% RSLogix 500 project I2P-Hands-On 4 - Adam Boczkiewicz.RSS, saved by version 10.00.00.00 %
PROJECT "UNTITLED"    % processor: Bul.1763 MicroLogix 1100 Series B %

PROGRAM FILES
  LAD 2   15 rungs

DATA FILES
  O0 OUTPUT  4 elements
  I1 INPUT  6 elements
  S2 STATUS  66 elements
  B3 BINARY  1 elements
  T4 TIMER  1 elements
  C5 COUNTER  1 elements
  R6 CONTROL  1 elements
  N7 INTEGER  1 elements
  F8 FLOAT  1 elements

LADDER 2
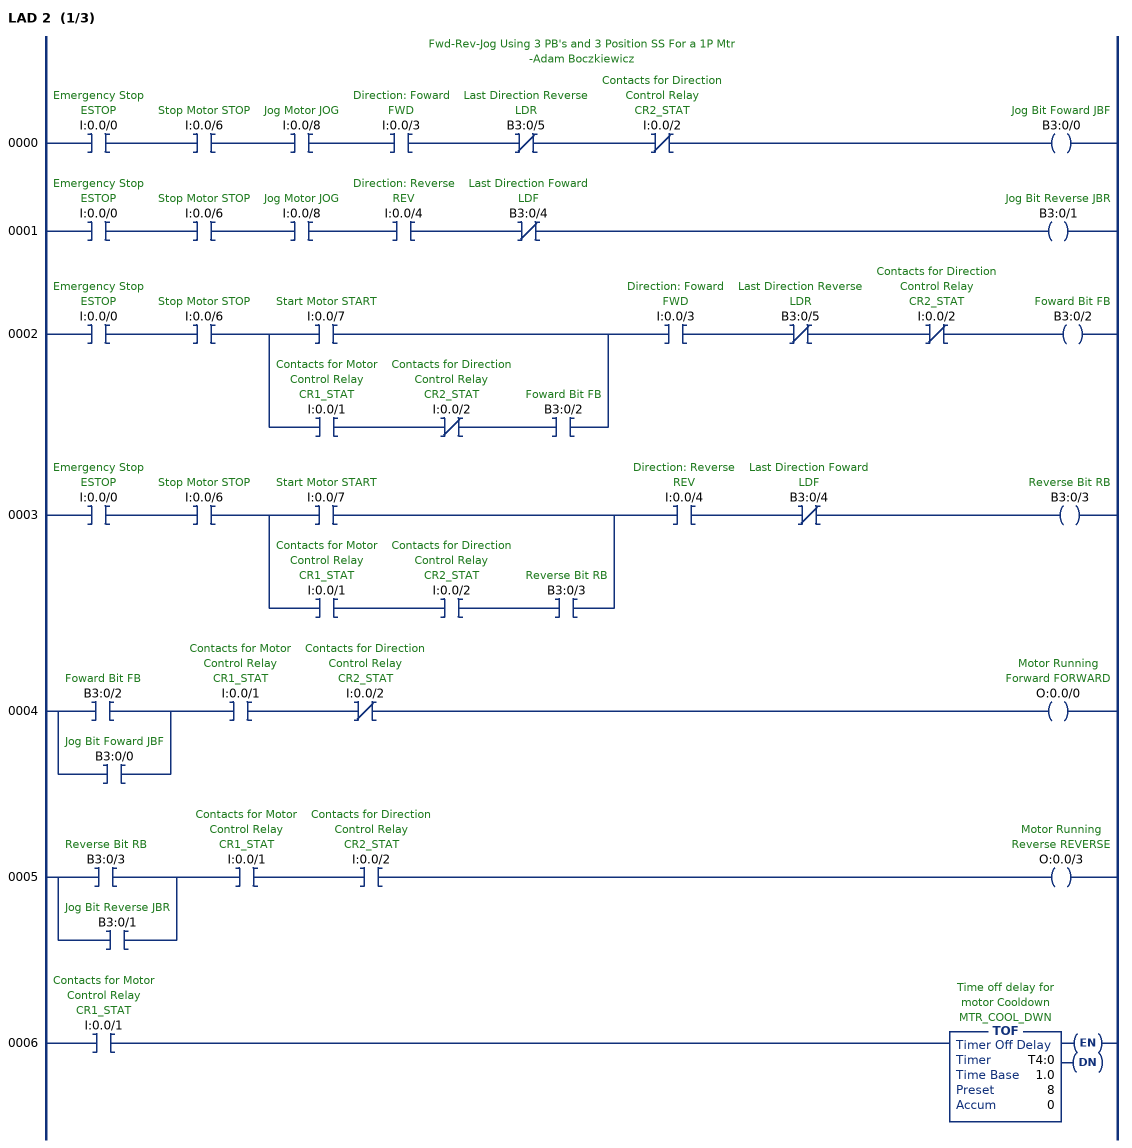
% Rung: 0 %
% Fwd-Rev-Jog Using 3 PB's and 3 Position SS For a 1P Mtr
% -Adam Boczkiewicz %
SOR XIC I:0.0/0 XIC I:0.0/6 XIC I:0.0/8 XIC I:0.0/3 XIO B3:0/5 XIO I:0.0/2 OTE B3:0/0 EOR
%   I:0.0/0  ESTOP  "Emergency Stop" %
%   I:0.0/6  STOP  "Stop Motor" %
%   I:0.0/8  JOG  "Jog Motor" %
%   I:0.0/3  FWD  "Direction: Foward" %
%   B3:0/5  LDR  "Last Direction Reverse" %
%   I:0.0/2  CR2_STAT  "Contacts for Direction Control Relay" %
%   B3:0/0  JBF  "Jog Bit Foward" %
% Rung: 1 %
SOR XIC I:0.0/0 XIC I:0.0/6 XIC I:0.0/8 XIC I:0.0/4 XIO B3:0/4 OTE B3:0/1 EOR
%   I:0.0/0  ESTOP  "Emergency Stop" %
%   I:0.0/6  STOP  "Stop Motor" %
%   I:0.0/8  JOG  "Jog Motor" %
%   I:0.0/4  REV  "Direction: Reverse" %
%   B3:0/4  LDF  "Last Direction Foward" %
%   B3:0/1  JBR  "Jog Bit Reverse" %
% Rung: 2 %
SOR XIC I:0.0/0 XIC I:0.0/6 BST XIC I:0.0/7 NXB XIC I:0.0/1 XIO I:0.0/2 XIC B3:0/2 BND XIC I:0.0/3 XIO B3:0/5 XIO I:0.0/2 OTE B3:0/2 EOR
%   I:0.0/0  ESTOP  "Emergency Stop" %
%   I:0.0/6  STOP  "Stop Motor" %
%   I:0.0/7  START  "Start Motor" %
%   I:0.0/1  CR1_STAT  "Contacts for Motor Control Relay" %
%   I:0.0/2  CR2_STAT  "Contacts for Direction Control Relay" %
%   B3:0/2  FB  "Foward Bit" %
%   I:0.0/3  FWD  "Direction: Foward" %
%   B3:0/5  LDR  "Last Direction Reverse" %
% Rung: 3 %
SOR XIC I:0.0/0 XIC I:0.0/6 BST XIC I:0.0/7 NXB XIC I:0.0/1 XIC I:0.0/2 XIC B3:0/3 BND XIC I:0.0/4 XIO B3:0/4 OTE B3:0/3 EOR
%   I:0.0/0  ESTOP  "Emergency Stop" %
%   I:0.0/6  STOP  "Stop Motor" %
%   I:0.0/7  START  "Start Motor" %
%   I:0.0/1  CR1_STAT  "Contacts for Motor Control Relay" %
%   I:0.0/2  CR2_STAT  "Contacts for Direction Control Relay" %
%   B3:0/3  RB  "Reverse Bit" %
%   I:0.0/4  REV  "Direction: Reverse" %
%   B3:0/4  LDF  "Last Direction Foward" %
% Rung: 4 %
SOR BST XIC B3:0/2 NXB XIC B3:0/0 BND XIC I:0.0/1 XIO I:0.0/2 OTE O:0.0/0 EOR
%   B3:0/2  FB  "Foward Bit" %
%   B3:0/0  JBF  "Jog Bit Foward" %
%   I:0.0/1  CR1_STAT  "Contacts for Motor Control Relay" %
%   I:0.0/2  CR2_STAT  "Contacts for Direction Control Relay" %
%   O:0.0/0  FORWARD  "Motor Running Forward" %
% Rung: 5 %
SOR BST XIC B3:0/3 NXB XIC B3:0/1 BND XIC I:0.0/1 XIC I:0.0/2 OTE O:0.0/3 EOR
%   B3:0/3  RB  "Reverse Bit" %
%   B3:0/1  JBR  "Jog Bit Reverse" %
%   I:0.0/1  CR1_STAT  "Contacts for Motor Control Relay" %
%   I:0.0/2  CR2_STAT  "Contacts for Direction Control Relay" %
%   O:0.0/3  REVERSE  "Motor Running Reverse" %
% Rung: 6 %
SOR XIC I:0.0/1 TOF T4:0 1.0 8 0 EOR
%   I:0.0/1  CR1_STAT  "Contacts for Motor Control Relay" %
%   T4:0  MTR_COOL_DWN  "Time off delay for motor Cooldown" %

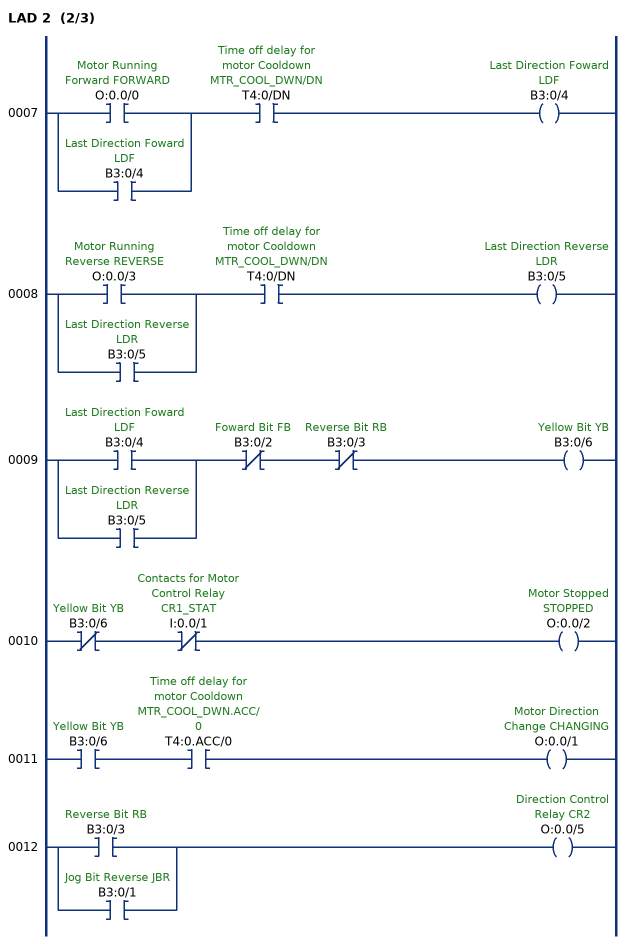
% Rung: 7 %
SOR BST XIC O:0.0/0 NXB XIC B3:0/4 BND XIC T4:0/DN OTE B3:0/4 EOR
%   O:0.0/0  FORWARD  "Motor Running Forward" %
%   B3:0/4  LDF  "Last Direction Foward" %
%   T4:0  MTR_COOL_DWN  "Time off delay for motor Cooldown" %
% Rung: 8 %
SOR BST XIC O:0.0/3 NXB XIC B3:0/5 BND XIC T4:0/DN OTE B3:0/5 EOR
%   O:0.0/3  REVERSE  "Motor Running Reverse" %
%   B3:0/5  LDR  "Last Direction Reverse" %
%   T4:0  MTR_COOL_DWN  "Time off delay for motor Cooldown" %
% Rung: 9 %
SOR BST XIC B3:0/4 NXB XIC B3:0/5 BND XIO B3:0/2 XIO B3:0/3 OTE B3:0/6 EOR
%   B3:0/4  LDF  "Last Direction Foward" %
%   B3:0/5  LDR  "Last Direction Reverse" %
%   B3:0/2  FB  "Foward Bit" %
%   B3:0/3  RB  "Reverse Bit" %
%   B3:0/6  YB  "Yellow Bit" %
% Rung: 10 %
SOR XIO B3:0/6 XIO I:0.0/1 OTE O:0.0/2 EOR
%   B3:0/6  YB  "Yellow Bit" %
%   I:0.0/1  CR1_STAT  "Contacts for Motor Control Relay" %
%   O:0.0/2  STOPPED  "Motor Stopped" %
% Rung: 11 %
SOR XIC B3:0/6 XIC T4:0.ACC/0 OTE O:0.0/1 EOR
%   B3:0/6  YB  "Yellow Bit" %
%   T4:0  MTR_COOL_DWN  "Time off delay for motor Cooldown" %
%   O:0.0/1  CHANGING  "Motor Direction Change" %
% Rung: 12 %
SOR BST XIC B3:0/3 NXB XIC B3:0/1 BND OTE O:0.0/5 EOR
%   B3:0/3  RB  "Reverse Bit" %
%   B3:0/1  JBR  "Jog Bit Reverse" %
%   O:0.0/5  CR2  "Direction Control Relay" %

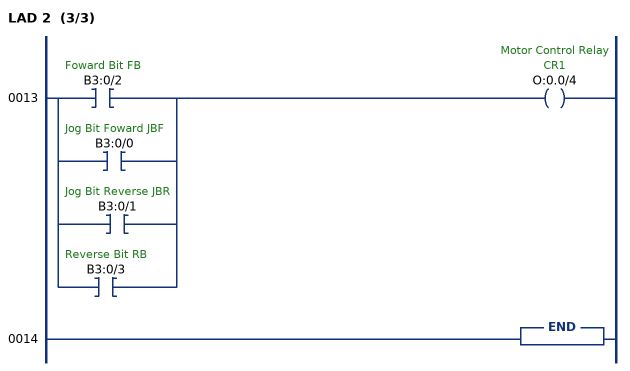
% Rung: 13 %
SOR BST XIC B3:0/2 NXB BST XIC B3:0/0 NXB BST XIC B3:0/1 NXB XIC B3:0/3 BND BND BND OTE O:0.0/4 EOR
%   B3:0/2  FB  "Foward Bit" %
%   B3:0/0  JBF  "Jog Bit Foward" %
%   B3:0/1  JBR  "Jog Bit Reverse" %
%   B3:0/3  RB  "Reverse Bit" %
%   O:0.0/4  CR1  "Motor Control Relay" %
% Rung: 14 %
SOR END EOR

OTHER DOCUMENTED ADDRESSES
  I  

DATA TABLE (non-zero values as saved)
DATA T4
% .PRE .ACC %
% T4:0 % 8 0
